// TIA Portal V17 export
// export: Created 2023-02-26T22:59:51.4230222Z, ExportSetting WithDefaults, DisplayName Totally Integrated Automation Portal, DisplayVersion V17, DisplayName TIA Portal Openness, DisplayVersion V17, DisplayName TIA Portal Version Control Interface, DisplayVersion V17, DisplayName TIA Portal Test Suite Advanced, DisplayVersion V17, DisplayName STEP 7 Professional, DisplayVersion V17, DisplayName SIMATIC Energy Suite, DisplayVersion V17, DisplayName STEP 7 Safety, DisplayVersion V17, DisplayName WinCC Professional, DisplayVersion V17
DATA_BLOCK "ERR_LostPackage_DB_3"   // DB28
VERSION : 0.1
// stored: AutoNumber true, InstanceOfName ERR_LostPackage, InstanceOfType FB
"ERR_LostPackage"
   // VAR_INPUT
   //    StartLine : Bool;
   //    StopLine : Bool;
   //    AutoMode : Bool;
   //    ResetButton : Bool;
   //    Di : Bool;
   //    Dj : Bool;
   //    FirstScan : Bool;
   //    "Time" : Time;
   // END_VAR
   // VAR_OUTPUT
   //    Error : Bool;
   // END_VAR
   // VAR
   //    S1 : Bool;
   //    S2 : Bool;
   //    S3 : Bool;
   //    t1 : Bool;
   //    P_ResetButton : Bool;
   //    IEC_Timer_0_Instance { ExternalAccessible := 'False'; ExternalVisible := 'False'; ExternalWritable := 'False'} : TON_TIME;
   // END_VAR
BEGIN
END_DATA_BLOCK
